KUKA KRL program: St1_Corner3.src, St1_Corner3.dat

--- St1_Corner3.src ---
&ACCESS RVEO
DEF  St1_Corner3 (lnActSt :IN,lnUseMillingTool :IN)
   INT lnActSt,lnUsedBase,lnUsedTool
   INT lnUseMillingTool,lnJobNr
   BOOL nbOK,lbTimeOut

   CONTINUE
   IF ($T1 OR $T2)THEN
      GLOBAL INTERRUPT DECL 3 WHEN $STOPMESS==TRUE DO IR_STOPM ( )
      INTERRUPT ON 3
      BAS (#INITMOV,0)
      lnActSt = 1
      PTP $POS_ACT
   ENDIF
   lnJobNr = gnJobNr3
   lnUsedBase = lnActSt + 10
   lnUsedTool = 20

   BASE_DATA[lnUsedBase] = BASE_DATA[lnActSt]:gfBaseShift[lnActSt]
   TOOL_DATA[lnUsedTool] = TOOL_DATA[11] :{X 0,Y 0,Z 0,A 0,B 0,C 0}

   MoveSettings(lnUsedBase, lnUsedTool, 100, 100)
   LIN lfPrePos[1] C_DIS

   MoveSettings(lnUsedBase, lnUsedTool, 100, 50)
   LIN lfPrePos[2] C_DIS
   REPEAT
      CONTINUE
   UNTIL DI_KEBFreqReached OR NOT WatchDog(gnTimerWatchDog, 5000)
   CONTINUE
   IF (NOT DI_KEBFreqReached ) THEN
      SpindleStop()
   ENDIF

    MoveToPrepos(lnActSt)
END

--- St1_Corner3.dat ---
&ACCESS RVEO
DEFDAT  St1_Corner3


DECL FRAME lfPrePos[3]
lfPrePos[1]={X -150.000,Y 0.0,Z 150.000,A 0.0,B 0.0,C 0.0}
lfPrePos[2]={X 0.0,Y 0.0,Z 0.0,A 0.0,B 0.0,C 0.0}
lfPrePos[3]={X 0.0,Y 0.0,Z 0.0,A 0.0,B 0.0,C 0.0}


DECL FRAME lfWorkPos[5]
lfWorkPos[1]={X -100.000,Y 0.0,Z 100.000,A 0.0,B 0.0,C 0.0}
lfWorkPos[2]={X 0.0,Y 0.0,Z 50.0000,A 0.0,B 0.0,C 0.0}
lfWorkPos[3]={X 0.0,Y 0.0,Z 25.0000,A 0.0,B 0.0,C 0.0}
lfWorkPos[4]={X -100.000,Y 0.0,Z 25.0000,A 0.0,B 0.0,C 0.0}
lfWorkPos[5]={X -150.000,Y 0.0,Z 150.000,A 0.0,B 0.0,C 0.0}


ENDDAT
